FUNCTION_BLOCK FB_InfoDecoupler
VAR_INPUT
	stInfoData 			: 		DUT_ST_InfoDataFB ;
END_VAR
VAR_OUTPUT
	sState 				: 		STRING ;
END_VAR
VAR
END_VAR

// Decouple FB's State
IF stInfoData.usiMapState 			=	0 THEN
				sState 				:= 	'Undefined' ;
	ELSIF stInfoData.usiMapState 	= 	1 THEN
				sState 				:= 	'RUN' ;
	ELSIF stInfoData.usiMapState 	= 	2 THEN
				sState 				:= 	'STOP' ;
ELSE
				sState 				:= 	'Unknown' ;
END_IF

// The Decouple FB Has No Diagnostic Byte to Decode

END_FUNCTION_BLOCK

(* stored: Version 1.1.0.1, ProductVersion 3.1.0.14
   POU FB_InfoDecoupler: Id {2ff0dfed-39a0-4e2e-a748-05636e7ae2f5} *)
